{attribute 'qualified_only'}
// BOOL: True/False

VAR_GLOBAL // Different modes true/false
	bRunning : BOOL;		// System running
	bManual : BOOL;			// Manual mode
	bAuto : BOOL;			// Auto mode
END_VAR

(* stored: Version 1.1.0.1
   GVL G_Mode: Id {a89507da-b50b-4379-9e9a-399fcb20c7fd} *)
